(* CoDeSys 2.3 export: GLOBAL_CONSTANTS.EXP *)

(* Global variable list: Global_Constants *)
VAR_GLOBAL CONSTANT
	MAXIMUM_HEATING_CIRCUITS_NUM : USINT := 3;
	(*Количество отопительных контуров*)

	MAX_UZ_NUM : USINT := 3;
	(*Количество частотных преобразователей UZ*)

	MAX_BOILERS_NUM : USINT := 3;
	(*Количество котлов*)

	MAX_K14_PUMPS_NUM : USINT := 3;
	(*Количество насосов К14*)

	MAX_K15_PUMPS_NUM : USINT := 2;
	(*Количество насосов К15*)

	MAX_K16_PUMPS_NUM : USINT := 2;
	(*Количество насосов К16*)
END_VAR
